INTERFACE I_HAL_DI

PROPERTY errId : uint
GET
END_GET
END_PROPERTY

PROPERTY xValue : bool
GET
END_GET
END_PROPERTY

END_INTERFACE

(* stored: Version 1.1.0.1, ProductVersion 3.1.4024.6
   Itf I_HAL_DI: Id {a6eb1073-59f8-02ab-208c-5166151e2101}
   Property errId: Id {1bbe2e54-8abf-0ed1-3f7f-39b7e3b042f5}
   Get Get: Id {847800c3-24c5-0ebd-05f5-572f57bc8076}
   Property xValue: Id {8d8cb2cd-132e-0e43-12e9-51f819d5cac3}
   Get Get: Id {340315db-132e-08d6-15bb-c078fee76ef2} *)
